FUNCTION Call_VisionSensor

instVisionSensorConveyor(PartPresent := PartDetectedVisionSensor,
													ValueCode := ReadPartCode,
													Error => ErrorVisionSensor);

END_FUNCTION

(* stored: Version 1.1.0.1
   POU Call_VisionSensor: Id {d50b5f90-bab1-414f-90c9-61597ce78258}, SpecialFunc None *)
